FUNCTION_BLOCK Fb_AnalogToReal_Conversion
VAR_INPUT
	iRawVal : UINT;
	iMinVal	: UINT;
	iMaxVal	: UINT;
	
END_VAR
VAR_OUTPUT
	lActualVal	: REAL;				//Actual converted value
	bError		: BOOL;
END_VAR           
VAR               
	lRangeHigh	: REAL := 32676;
	lRawVal 	: REAL;
	lMinVal		: REAL;
	lMaxVal		: REAL;
END_VAR

lRawVal	:=UINT_TO_REAL(iRawVal);
lMinVal	:=UINT_TO_REAL(iMinVal);
lMaxVal	:=UINT_TO_REAL(iMaxVal);

IF iRawVal<=0 THEN
	lActualVal:=0;
END_IF

IF NOT iRawVal>0 AND iRawVal<=lRangeHigh THEN	
	lActualVal := ((lMaxVal-lMinVal)/(lRangeHigh-0))*lRawVal+lMinVal;
	bError:=FALSE;
ELSE
	bError:=TRUE;	
END_IF

METHOD Error_Check : BOOL
VAR_INPUT
END_VAR
END_METHOD

METHOD RawToRealConversion : BOOL
VAR_INPUT
END_VAR
END_METHOD

END_FUNCTION_BLOCK

(* stored: Version 1.1.0.1, ProductVersion 3.1.4024.12
   POU Fb_AnalogToReal_Conversion: Id {420ab8ec-5ef5-487b-ab0f-52224fffdeca}, SpecialFunc None
   Method Error_Check: Id {8952912d-742b-42c7-aa0e-5d176a00600a}
   Method RawToRealConversion: Id {466f3449-b983-4009-942e-d1e81a74a8c4} *)
